FUNCTION_BLOCK FB_FileRingBufferToDB
VAR_INPUT
	udiNovRam_BufferIndex:UDINT;
	udiFile_Index:UDINT;
	dataType:DINT;
END_VAR
VAR_IN_OUT
	NovRamData:ST_NovRam;
END_VAR

IF dataType = E_DB_StructureType.AlarmHistory THEN
	M_AlarmHistory(udiNovRam_BufferIndex:=udiNovRam_BufferIndex,udiFile_Index:=udiFile_Index);
ELSIF dataType = E_DB_StructureType.ProductionHistory THEN
	M_ProductionHistory(udiNovRam_BufferIndex:=udiNovRam_BufferIndex,udiFile_Index:=udiFile_Index);
ELSIF dataType = E_DB_StructureType.ProductionReport THEN
	M_ProductionReport(udiNovRam_BufferIndex:=udiNovRam_BufferIndex,udiFile_Index:=udiFile_Index);
ELSIF dataType = E_DB_StructureType.ProductionSummary THEN
	M_ProductionSummary(udiNovRam_BufferIndex:=udiNovRam_BufferIndex,udiFile_Index:=udiFile_Index);
ELSIF dataType = E_DB_StructureType.SoDuration THEN
	M_SoDuration(udiNovRam_BufferIndex:=udiNovRam_BufferIndex,udiFile_Index:=udiFile_Index);
ELSIF dataType = E_DB_StructureType.StopCount THEN
	M_StopCount(udiNovRam_BufferIndex:=udiNovRam_BufferIndex,udiFile_Index:=udiFile_Index);
ELSIF dataType = E_DB_StructureType.RegularCheckResults THEN
	M_RegularCheckResults(udiNovRam_BufferIndex:=udiNovRam_BufferIndex,udiFile_Index:=udiFile_Index);
END_IF

METHOD M_AlarmHistory : BOOL
VAR_INPUT
	
	//udiFileNo:UDINT;
	udiNovRam_BufferIndex:UDINT;
	udiFile_Index:UDINT;
END_VAR
VAR_INST
	arrDataFromFile:ARRAY[0..GVL.arrArrayLength[E_DB_StructureType.AlarmHistory]-1] OF ST_AlarmInfo_DB_save;//small
	DataToDB:ST_AlarmInfo_DB;//large
	AnalizeIndex:UDINT;//should be kept by NovRam
	iStep:INT;
	i:UDINT;
	fbFileRingBuffer: FB_FileRingBuffer := ( sNetId     := '',
                                             sPathName  := '',
                                             ePath      := PATH_GENERIC,
                                             nID        := 1,
                                             cbBuffer   := gvl.arrFileRingBufferSize[E_DB_StructureType.AlarmHistory], //5MB(5*10^6Bytes)
                                             bOverwrite := FALSE,
                                             pWriteBuff := 0,
                                             cbWriteLen := 0,
                                             pReadBuff  := 0,
                                             cbReadLen  := 0,
                                             tTimeout   := T#1S );
	bBusy:BOOL;
	bError:BOOL;
	nErrID:UDINT;
	stHeader:ST_FileRBufferHead;
    //loadData  : ARRAY[0..511] OF BYTE :=[512(0)];
    //cbLoad    : UDINT;
	
	fileName: STRING(255);
	eStrIndex:DINT;
	fbAlarmHistory_DB		: FB_AlarmHistory_DB;
END_VAR
//Config
eStrIndex:=E_DB_StructureType.AlarmHistory;

fbFileRingBuffer(sPathName:=fileName
				,bBusy=>bBusy,bError=>bError,nErrID=>nErrID
				,stHeader=>stHeader);
//DB_Test
fbAlarmHistory_DB(udiDBID:=1);

CASE iStep OF
	0://check if file full 
		IF NovRamData.arrFileRingBuffer_Status[eStrIndex].bFileFull[udiNovRam_BufferIndex][udiFile_Index] = TRUE//file full = should work 
		THEN
			
			fileName:=M_GetFileName(structureType:=eStrIndex
									,udiNovRam_BufferIndex:=udiNovRam_BufferIndex
									,udiFile_Index:=udiFile_Index);
			
			iStep:=100;
		END_IF
	100:// Open file
		
		AnalizeIndex:=0;
		fbFileRingBuffer.A_Open();
		
		iStep:=200;
	200://wait done / read head
		IF NOT fbFileRingBuffer.bBusy AND NOT fbFileRingBuffer.bError THEN
			
			fbFileRingBuffer.A_GetHead(pReadBuff := ADR(arrDataFromFile), cbReadLen := SIZEOF(arrDataFromFile));
			
			iStep:=300;
		END_IF
	300://wait done / take data from array
		IF NOT fbFileRingBuffer.bBusy AND NOT fbFileRingBuffer.bError THEN
			
			M_ST_AlarmHistory_Extract(Input:=arrDataFromFile[AnalizeIndex],Output=>DataToDB);
			//DataToDB:=arrDataFromFile[AnalizeIndex];
			
			iStep:=310;
		ELSIF NOT fbFileRingBuffer.bBusy AND fbFileRingBuffer.bError THEN//Empty
			iStep:=600;
		END_IF
	310:// write to DB
	
		IF fbAlarmHistory_DB.M_Upload(stAlarmInfo:=DataToDB) THEN
			iStep:=320;
		END_IF
		
	320://wait done
		
		IF NOT fbAlarmHistory_DB.bError THEN//write OK
		
			AnalizeIndex:=AnalizeIndex+1;
			
			iStep:=330;
			
		ELSE//write failed need to write to log
			;
		END_IF
		
	330://Check if all data in array Analized
		IF AnalizeIndex < GVL.arrArrayLength[eStrIndex]-1 THEN//not done
			iStep:=300;//go back
		ELSE//array data done
			iStep:=400;//complete this array
		END_IF
		
	400://wait done / remove Head
	
		fbFileRingBuffer.A_RemoveHead(pReadBuff := ADR(arrDataFromFile), cbReadLen := SIZEOF(arrDataFromFile));
		
		iStep:=500;
		
	500://wait done / check if all data got?
		IF NOT fbFileRingBuffer.bBusy AND NOT fbFileRingBuffer.bError THEN
			IF stHeader.nCount > 0 THEN
				iStep:=100;//Go Back
			ELSE
				iStep:=600;//finish
			END_IF
		END_IF
	600://reset file
	
		fbFileRingBuffer.A_Reset();
		
		iStep:=700;
		
	700://wait done / close file
		IF NOT fbFileRingBuffer.bBusy AND NOT fbFileRingBuffer.bError THEN
			
			fbFileRingBuffer.A_Close();
			
			iStep:=800;
		END_IF
	800://wait done
		IF NOT fbFileRingBuffer.bBusy AND NOT fbFileRingBuffer.bError THEN
			
			NovRamData.arrFileRingBuffer_Status[eStrIndex].bFileFull[udiNovRam_BufferIndex][udiFile_Index]:=FALSE;
			
			iStep:=0;
			
		END_IF
		
	
END_CASE
END_METHOD

METHOD M_GetFileName : STRING(255)
VAR_INPUT
	structureType:DINT;
	udiNovRam_BufferIndex:UDINT;
	udiFile_Index:UDINT;
END_VAR
VAR
	tempString:STRING(255);
	tempString2:STRING(255);
	tempFileNo:UDINT;
END_VAR
IF structureType=E_DB_StructureType.AlarmHistory THEN
	tempString:=CONCAT(gvl.arrfileFolder[structureType],'AlarmHistory');
ELSIF structureType=E_DB_StructureType.ProductionHistory THEN
	tempString:=CONCAT(gvl.arrfileFolder[structureType],'ProductionHistory');
ELSIF structureType=E_DB_StructureType.ProductionReport THEN
	tempString:=CONCAT(gvl.arrfileFolder[structureType],'ProductionReport');
ELSIF structureType=E_DB_StructureType.ProductionSummary THEN
	tempString:=CONCAT(gvl.arrfileFolder[structureType],'ProductionSummary');
ELSIF structureType=E_DB_StructureType.SoDuration THEN
	tempString:=CONCAT(gvl.arrfileFolder[structureType],'SoDuration');
ELSIF structureType=E_DB_StructureType.StopCount THEN
	tempString:=CONCAT(gvl.arrfileFolder[structureType],'StopCount');
ELSIF structureType=E_DB_StructureType.RegularCheckResults THEN
	tempString:=CONCAT(gvl.arrfileFolder[structureType],'RegularCheckResults');
END_IF

tempFileNo:=(udiNovRam_BufferIndex) * GVL.FileRingBufferRatio + (udiFile_Index + 1);
tempString2:=CONCAT(tempString,UDINT_TO_STRING(tempFileNo));
M_GetFileName:=CONCAT(tempString2,'.dat');
END_METHOD

{warning 'add method implementation '}
METHOD M_ProductionHistory : BOOL
VAR_INPUT
	
	//udiFileNo:UDINT;
	udiNovRam_BufferIndex:UDINT;
	udiFile_Index:UDINT;
END_VAR
VAR_INST
	arrDataFromFile:ARRAY[0..GVL.arrArrayLength[E_DB_StructureType.ProductionHistory]-1] OF ST_PHI_GroupData_DB;//small
	DataToDB:ST_PHI_GroupData_DB;//large
	AnalizeIndex:UDINT;//should be kept by NovRam
	iStep:INT;
	i:UDINT;
	fbFileRingBuffer: FB_FileRingBuffer := ( sNetId     := '',
                                             sPathName  := '',
                                             ePath      := PATH_GENERIC,
                                             nID        := 1,
                                             cbBuffer   := gvl.arrFileRingBufferSize[E_DB_StructureType.ProductionHistory], //5MB(5*10^6Bytes)
                                             bOverwrite := FALSE,
                                             pWriteBuff := 0,
                                             cbWriteLen := 0,
                                             pReadBuff  := 0,
                                             cbReadLen  := 0,
                                             tTimeout   := T#1S );
	bBusy:BOOL;
	bError:BOOL;
	nErrID:UDINT;
	stHeader:ST_FileRBufferHead;
    //loadData  : ARRAY[0..511] OF BYTE :=[512(0)];
    //cbLoad    : UDINT;
	
	fileName: STRING(255);
	eStrIndex:DINT;
	
	//DB
	fbProductionHistoryInspection_DB		: FB_ProductionHistoryInspection_DB;
	PHI_GroupData_DB : ST_PHI_GroupData_DB;
END_VAR
//Config
eStrIndex:=E_DB_StructureType.ProductionHistory;

fbFileRingBuffer(sPathName:=fileName
				,bBusy=>bBusy,bError=>bError,nErrID=>nErrID
				,stHeader=>stHeader);
				
//DB_Test
fbProductionHistoryInspection_DB(udiDBID:=1);

CASE iStep OF
	0://check if file full 
		IF NovRamData.arrFileRingBuffer_Status[eStrIndex].bFileFull[udiNovRam_BufferIndex][udiFile_Index] = TRUE//file full = should work 
		THEN
			
			fileName:=M_GetFileName(structureType:=eStrIndex
									,udiNovRam_BufferIndex:=udiNovRam_BufferIndex
									,udiFile_Index:=udiFile_Index);
			
			iStep:=100;
		END_IF
	100:// Open file
		
		AnalizeIndex:=0;
		fbFileRingBuffer.A_Open();
		
		iStep:=200;
	200://wait done / read head
		IF NOT fbFileRingBuffer.bBusy AND NOT fbFileRingBuffer.bError THEN
			
			fbFileRingBuffer.A_GetHead(pReadBuff := ADR(arrDataFromFile), cbReadLen := SIZEOF(arrDataFromFile));
			
			iStep:=300;
		END_IF
	300://wait done / take data from array
		IF NOT fbFileRingBuffer.bBusy AND NOT fbFileRingBuffer.bError THEN
			
			M_ST_ProductionHistory_Extract(Input:=arrDataFromFile[AnalizeIndex],Output=>DataToDB);
			//DataToDB:=arrDataFromFile[AnalizeIndex];
			
			iStep:=310;
		ELSIF NOT fbFileRingBuffer.bBusy AND fbFileRingBuffer.bError THEN//Empty
			iStep:=600;
		END_IF
	310:// write to DB
	
		IF fbProductionHistoryInspection_DB.M_Upload(stPHI:=DataToDB) THEN
			iStep:=320;
		END_IF
		
	320://wait done
		
		IF NOT fbProductionHistoryInspection_DB.bError THEN//write OK
		
			AnalizeIndex:=AnalizeIndex+1;
			
			iStep:=330;
			
		ELSE//write failed need to write to log
			;
		END_IF
		
	330://Check if all data in array Analized
		IF AnalizeIndex < GVL.arrArrayLength[eStrIndex]-1 THEN//not done
			iStep:=300;//go back
		ELSE//array data done
			iStep:=400;//complete this array
		END_IF
		
	400://wait done / remove Head
	
		fbFileRingBuffer.A_RemoveHead(pReadBuff := ADR(arrDataFromFile), cbReadLen := SIZEOF(arrDataFromFile));
		
		iStep:=500;
		
	500://wait done / check if all data got?
		IF NOT fbFileRingBuffer.bBusy AND NOT fbFileRingBuffer.bError THEN
			IF stHeader.nCount > 0 THEN
				iStep:=100;//Go Back
			ELSE
				iStep:=600;//finish
			END_IF
		END_IF
	600://reset file
	
		fbFileRingBuffer.A_Reset();
		
		iStep:=700;
		
	700://wait done / close file
		IF NOT fbFileRingBuffer.bBusy AND NOT fbFileRingBuffer.bError THEN
			
			fbFileRingBuffer.A_Close();
			
			iStep:=800;
		END_IF
	800://wait done
		IF NOT fbFileRingBuffer.bBusy AND NOT fbFileRingBuffer.bError THEN
			
			NovRamData.arrFileRingBuffer_Status[eStrIndex].bFileFull[udiNovRam_BufferIndex][udiFile_Index]:=FALSE;
			
			iStep:=0;
			
		END_IF
		
	
END_CASE
END_METHOD

METHOD M_ProductionReport : BOOL
VAR_INPUT
	
	//udiFileNo:UDINT;
	udiNovRam_BufferIndex:UDINT;
	udiFile_Index:UDINT;
END_VAR
VAR_INST
	arrDataFromFile:ARRAY[0..GVL.arrArrayLength[E_DB_StructureType.ProductionReport]-1] OF ST_OEE_ProductionReport;//small
	DataToDB:ST_OEE_ProductionReport;//large
	AnalizeIndex:UDINT;//should be kept by NovRam
	iStep:INT;
	i:UDINT;
	fbFileRingBuffer: FB_FileRingBuffer := ( sNetId     := '',
                                             sPathName  := '',
                                             ePath      := PATH_GENERIC,
                                             nID        := 1,
                                             cbBuffer   := gvl.arrFileRingBufferSize[E_DB_StructureType.ProductionReport], //5MB(5*10^6Bytes)
                                             bOverwrite := FALSE,
                                             pWriteBuff := 0,
                                             cbWriteLen := 0,
                                             pReadBuff  := 0,
                                             cbReadLen  := 0,
                                             tTimeout   := T#1S );
	bBusy:BOOL;
	bError:BOOL;
	nErrID:UDINT;
	stHeader:ST_FileRBufferHead;
    //loadData  : ARRAY[0..511] OF BYTE :=[512(0)];
    //cbLoad    : UDINT;
	
	fileName: STRING(255);
	eStrIndex:DINT;
	fbOEE_ProductionReport_DB:FB_OEE_ProductionReport_DB;
END_VAR
//Config
eStrIndex:=E_DB_StructureType.ProductionReport;

fbFileRingBuffer(sPathName:=fileName
				,bBusy=>bBusy,bError=>bError,nErrID=>nErrID
				,stHeader=>stHeader);
				
CASE iStep OF
	0://check if file full 
		IF NovRamData.arrFileRingBuffer_Status[eStrIndex].bFileFull[udiNovRam_BufferIndex][udiFile_Index] = TRUE//file full = should work 
		THEN
			
			fileName:=M_GetFileName(structureType:=eStrIndex
									,udiNovRam_BufferIndex:=udiNovRam_BufferIndex
									,udiFile_Index:=udiFile_Index);
			
			iStep:=100;
		END_IF
	100:// Open file
		
		AnalizeIndex:=0;
		fbFileRingBuffer.A_Open();
		
		iStep:=200;
	200://wait done / read head
		IF NOT fbFileRingBuffer.bBusy AND NOT fbFileRingBuffer.bError THEN
			
			fbFileRingBuffer.A_GetHead(pReadBuff := ADR(arrDataFromFile), cbReadLen := SIZEOF(arrDataFromFile));
			
			iStep:=300;
		END_IF
	300://wait done / take data from array
		IF NOT fbFileRingBuffer.bBusy AND NOT fbFileRingBuffer.bError THEN
			
			M_ST_ProductionReport_Extract(Input:=arrDataFromFile[AnalizeIndex],Output=>DataToDB);
			//DataToDB:=arrDataFromFile[AnalizeIndex];
			
			iStep:=310;
		ELSIF NOT fbFileRingBuffer.bBusy AND fbFileRingBuffer.bError THEN//Empty
			iStep:=600;
		END_IF
	310:// write to DB
	
		IF fbOEE_ProductionReport_DB.M_Upload(stOeeProductionReport:=DataToDB) THEN
			iStep:=320;
		END_IF
		
	320://wait done
		
			IF NOT fbOEE_ProductionReport_DB.bError THEN//write OK
			
				AnalizeIndex:=AnalizeIndex+1;
				
				iStep:=330;
				
			ELSE//write failed need to write to log
				;
			END_IF
		
		
	330://Check if all data in array Analized
		IF AnalizeIndex < GVL.arrArrayLength[eStrIndex]-1 THEN//not done
			iStep:=300;//go back
		ELSE//array data done
			iStep:=400;//complete this array
		END_IF
		
	400://wait done / remove Head
	
		fbFileRingBuffer.A_RemoveHead(pReadBuff := ADR(arrDataFromFile), cbReadLen := SIZEOF(arrDataFromFile));
		
		iStep:=500;
		
	500://wait done / check if all data got?
		IF NOT fbFileRingBuffer.bBusy AND NOT fbFileRingBuffer.bError THEN
			IF stHeader.nCount > 0 THEN
				iStep:=100;//Go Back
			ELSE
				iStep:=600;//finish
			END_IF
		END_IF
	600://reset file
	
		fbFileRingBuffer.A_Reset();
		
		iStep:=700;
		
	700://wait done / close file
		IF NOT fbFileRingBuffer.bBusy AND NOT fbFileRingBuffer.bError THEN
			
			fbFileRingBuffer.A_Close();
			
			iStep:=800;
		END_IF
	800://wait done
		IF NOT fbFileRingBuffer.bBusy AND NOT fbFileRingBuffer.bError THEN
			
			NovRamData.arrFileRingBuffer_Status[eStrIndex].bFileFull[udiNovRam_BufferIndex][udiFile_Index]:=FALSE;
			
			iStep:=0;
			
		END_IF
		
	
END_CASE
END_METHOD

METHOD M_ProductionSummary : BOOL
VAR_INPUT
	
	//udiFileNo:UDINT;
	udiNovRam_BufferIndex:UDINT;
	udiFile_Index:UDINT;
END_VAR
VAR_INST
	arrDataFromFile:ARRAY[0..GVL.arrArrayLength[E_DB_StructureType.ProductionSummary]-1] OF ST_OEE_ProductionSummary;//small
	DataToDB:ST_OEE_ProductionSummary;//large
	AnalizeIndex:UDINT;//should be kept by NovRam
	iStep:INT;
	i:UDINT;
	fbFileRingBuffer: FB_FileRingBuffer := ( sNetId     := '',
                                             sPathName  := '',
                                             ePath      := PATH_GENERIC,
                                             nID        := 1,
                                             cbBuffer   := gvl.arrFileRingBufferSize[E_DB_StructureType.ProductionSummary], //5MB(5*10^6Bytes)
                                             bOverwrite := FALSE,
                                             pWriteBuff := 0,
                                             cbWriteLen := 0,
                                             pReadBuff  := 0,
                                             cbReadLen  := 0,
                                             tTimeout   := T#1S );
	bBusy:BOOL;
	bError:BOOL;
	nErrID:UDINT;
	stHeader:ST_FileRBufferHead;
    //loadData  : ARRAY[0..511] OF BYTE :=[512(0)];
    //cbLoad    : UDINT;
	
	fileName: STRING(255);
	eStrIndex:DINT;
	fbOEE_ProductionSummary_DB:FB_OEE_ProductionSummary_DB;
END_VAR
//Config
eStrIndex:=E_DB_StructureType.ProductionSummary;

fbFileRingBuffer(sPathName:=fileName
				,bBusy=>bBusy,bError=>bError,nErrID=>nErrID
				,stHeader=>stHeader);
				
CASE iStep OF
	0://check if file full 
		IF NovRamData.arrFileRingBuffer_Status[eStrIndex].bFileFull[udiNovRam_BufferIndex][udiFile_Index] = TRUE//file full = should work 
		THEN
			
			fileName:=M_GetFileName(structureType:=eStrIndex
									,udiNovRam_BufferIndex:=udiNovRam_BufferIndex
									,udiFile_Index:=udiFile_Index);
			
			iStep:=100;
		END_IF
	100:// Open file
		
		AnalizeIndex:=0;
		fbFileRingBuffer.A_Open();
		
		iStep:=200;
	200://wait done / read head
		IF NOT fbFileRingBuffer.bBusy AND NOT fbFileRingBuffer.bError THEN
			
			fbFileRingBuffer.A_GetHead(pReadBuff := ADR(arrDataFromFile), cbReadLen := SIZEOF(arrDataFromFile));
			
			iStep:=300;
		END_IF
	300://wait done / take data from array
		IF NOT fbFileRingBuffer.bBusy AND NOT fbFileRingBuffer.bError THEN
			
			M_ST_ProductionSummary_Extract(Input:=arrDataFromFile[AnalizeIndex],Output=>DataToDB);
			//DataToDB:=arrDataFromFile[AnalizeIndex];
			
			iStep:=310;
		ELSIF NOT fbFileRingBuffer.bBusy AND fbFileRingBuffer.bError THEN//Empty
			iStep:=600;
		END_IF
	310:// write to DB
	
		IF fbOEE_ProductionSummary_DB.M_Upload(stOEEProductionSummary:=DataToDB) THEN
			iStep:=320;
		END_IF
		
	320://wait done
		
			IF NOT fbOEE_ProductionSummary_DB.bError THEN//write OK
			
				AnalizeIndex:=AnalizeIndex+1;
				
				iStep:=330;
				
			ELSE//write failed need to write to log
				;
			END_IF
		
		
	330://Check if all data in array Analized
		IF AnalizeIndex < GVL.arrArrayLength[eStrIndex]-1 THEN//not done
			iStep:=300;//go back
		ELSE//array data done
			iStep:=400;//complete this array
		END_IF
		
	400://wait done / remove Head
	
		fbFileRingBuffer.A_RemoveHead(pReadBuff := ADR(arrDataFromFile), cbReadLen := SIZEOF(arrDataFromFile));
		
		iStep:=500;
		
	500://wait done / check if all data got?
		IF NOT fbFileRingBuffer.bBusy AND NOT fbFileRingBuffer.bError THEN
			IF stHeader.nCount > 0 THEN
				iStep:=100;//Go Back
			ELSE
				iStep:=600;//finish
			END_IF
		END_IF
	600://reset file
	
		fbFileRingBuffer.A_Reset();
		
		iStep:=700;
		
	700://wait done / close file
		IF NOT fbFileRingBuffer.bBusy AND NOT fbFileRingBuffer.bError THEN
			
			fbFileRingBuffer.A_Close();
			
			iStep:=800;
		END_IF
	800://wait done
		IF NOT fbFileRingBuffer.bBusy AND NOT fbFileRingBuffer.bError THEN
			
			NovRamData.arrFileRingBuffer_Status[eStrIndex].bFileFull[udiNovRam_BufferIndex][udiFile_Index]:=FALSE;
			
			iStep:=0;
			
		END_IF
		
	
END_CASE
END_METHOD

METHOD M_RegularCheckResults : BOOL
VAR_INPUT
	
	//udiFileNo:UDINT;
	udiNovRam_BufferIndex:UDINT;
	udiFile_Index:UDINT;
END_VAR
VAR_INST
	arrDataFromFile:ARRAY[0..GVL.arrArrayLength[E_DB_StructureType.RegularCheckResults]-1] OF ST_RegularCheck_Results;//small
	DataToDB:ST_RegularCheck_Results;//large
	AnalizeIndex:UDINT;//should be kept by NovRam
	iStep:INT;
	i:UDINT;
	fbFileRingBuffer: FB_FileRingBuffer := ( sNetId     := '',
                                             sPathName  := '',
                                             ePath      := PATH_GENERIC,
                                             nID        := 1,
                                             cbBuffer   := gvl.arrFileRingBufferSize[E_DB_StructureType.RegularCheckResults], //5MB(5*10^6Bytes)
                                             bOverwrite := FALSE,
                                             pWriteBuff := 0,
                                             cbWriteLen := 0,
                                             pReadBuff  := 0,
                                             cbReadLen  := 0,
                                             tTimeout   := T#1S );
	bBusy:BOOL;
	bError:BOOL;
	nErrID:UDINT;
	stHeader:ST_FileRBufferHead;
    //loadData  : ARRAY[0..511] OF BYTE :=[512(0)];
    //cbLoad    : UDINT;
	
	fileName: STRING(255);
	eStrIndex:DINT;
	fbRegular_Check_Results_DB:FB_Regular_Check_Results_DB;
END_VAR
//Config
eStrIndex:=E_DB_StructureType.RegularCheckResults;

fbFileRingBuffer(sPathName:=fileName
				,bBusy=>bBusy,bError=>bError,nErrID=>nErrID
				,stHeader=>stHeader);
				
CASE iStep OF
	0://check if file full 
		IF NovRamData.arrFileRingBuffer_Status[eStrIndex].bFileFull[udiNovRam_BufferIndex][udiFile_Index] = TRUE//file full = should work 
		THEN
			
			fileName:=M_GetFileName(structureType:=eStrIndex
									,udiNovRam_BufferIndex:=udiNovRam_BufferIndex
									,udiFile_Index:=udiFile_Index);
			
			iStep:=100;
		END_IF
	100:// Open file
		
		AnalizeIndex:=0;
		fbFileRingBuffer.A_Open();
		
		iStep:=200;
	200://wait done / read head
		IF NOT fbFileRingBuffer.bBusy AND NOT fbFileRingBuffer.bError THEN
			
			fbFileRingBuffer.A_GetHead(pReadBuff := ADR(arrDataFromFile), cbReadLen := SIZEOF(arrDataFromFile));
			
			iStep:=300;
		END_IF
	300://wait done / take data from array
		IF NOT fbFileRingBuffer.bBusy AND NOT fbFileRingBuffer.bError THEN
			
			M_ST_RegularCheckResults_Extract(Input:=arrDataFromFile[AnalizeIndex],Output=>DataToDB);
			//DataToDB:=arrDataFromFile[AnalizeIndex];
								
			iStep:=310;
		ELSIF NOT fbFileRingBuffer.bBusy AND fbFileRingBuffer.bError THEN//Empty
			iStep:=600;
		END_IF
	310:// write to DB
		
		IF fbRegular_Check_Results_DB.M_Upload(stRcResults:=DataToDB) THEN
			iStep:=320;
		END_IF
		
	320://wait done
		
		IF NOT fbRegular_Check_Results_DB.bError THEN//write OK
		
			AnalizeIndex:=AnalizeIndex+1;
			
			iStep:=330;
			
		ELSE//write failed need to write to log
			;
		END_IF
		
	330://Check if all data in array Analized
		IF AnalizeIndex < GVL.arrArrayLength[eStrIndex]-1 THEN//not done
			iStep:=300;//go back
		ELSE//array data done
			iStep:=400;//complete this array
		END_IF
		
	400://wait done / remove Head
	
		fbFileRingBuffer.A_RemoveHead(pReadBuff := ADR(arrDataFromFile), cbReadLen := SIZEOF(arrDataFromFile));
		
		iStep:=500;
		
	500://wait done / check if all data got?
		IF NOT fbFileRingBuffer.bBusy AND NOT fbFileRingBuffer.bError THEN
			IF stHeader.nCount > 0 THEN
				iStep:=100;//Go Back
			ELSE
				iStep:=600;//finish
			END_IF
		END_IF
	600://reset file
	
		fbFileRingBuffer.A_Reset();
		
		iStep:=700;
		
	700://wait done / close file
		IF NOT fbFileRingBuffer.bBusy AND NOT fbFileRingBuffer.bError THEN
			
			fbFileRingBuffer.A_Close();
			
			iStep:=800;
		END_IF
	800://wait done
		IF NOT fbFileRingBuffer.bBusy AND NOT fbFileRingBuffer.bError THEN
			
			NovRamData.arrFileRingBuffer_Status[eStrIndex].bFileFull[udiNovRam_BufferIndex][udiFile_Index]:=FALSE;
			
			iStep:=0;
			
		END_IF
		
	
END_CASE
END_METHOD

METHOD M_SoDuration : BOOL
VAR_INPUT
	
	//udiFileNo:UDINT;
	udiNovRam_BufferIndex:UDINT;
	udiFile_Index:UDINT;
END_VAR
VAR_INST
	arrDataFromFile:ARRAY[0..GVL.arrArrayLength[E_DB_StructureType.SoDuration]-1] OF ST_SoDuration;//small
	DataToDB:ST_SoDuration;//large
	AnalizeIndex:UDINT;//should be kept by NovRam
	iStep:INT;
	i:UDINT;
	fbFileRingBuffer: FB_FileRingBuffer := ( sNetId     := '',
                                             sPathName  := '',
                                             ePath      := PATH_GENERIC,
                                             nID        := 1,
                                             cbBuffer   := gvl.arrFileRingBufferSize[E_DB_StructureType.ProductionSummary], //5MB(5*10^6Bytes)
                                             bOverwrite := FALSE,
                                             pWriteBuff := 0,
                                             cbWriteLen := 0,
                                             pReadBuff  := 0,
                                             cbReadLen  := 0,
                                             tTimeout   := T#1S );
	bBusy:BOOL;
	bError:BOOL;
	nErrID:UDINT;
	stHeader:ST_FileRBufferHead;
    //loadData  : ARRAY[0..511] OF BYTE :=[512(0)];
    //cbLoad    : UDINT;
	
	fileName: STRING(255);
	eStrIndex:DINT;
	fbSoDuration_DB:FB_SoDuration_DB;
	
END_VAR
//Config
eStrIndex:=E_DB_StructureType.SoDuration;

fbFileRingBuffer(sPathName:=fileName
				,bBusy=>bBusy,bError=>bError,nErrID=>nErrID
				,stHeader=>stHeader);
				
CASE iStep OF
	0://check if file full 
		IF NovRamData.arrFileRingBuffer_Status[eStrIndex].bFileFull[udiNovRam_BufferIndex][udiFile_Index] = TRUE//file full = should work 
		THEN
			
			fileName:=M_GetFileName(structureType:=eStrIndex
									,udiNovRam_BufferIndex:=udiNovRam_BufferIndex
									,udiFile_Index:=udiFile_Index);
			
			iStep:=100;
		END_IF
	100:// Open file
		
		AnalizeIndex:=0;
		fbFileRingBuffer.A_Open();
		
		iStep:=200;
	200://wait done / read head
		IF NOT fbFileRingBuffer.bBusy AND NOT fbFileRingBuffer.bError THEN
			
			fbFileRingBuffer.A_GetHead(pReadBuff := ADR(arrDataFromFile), cbReadLen := SIZEOF(arrDataFromFile));
			
			iStep:=300;
		END_IF
	300://wait done / take data from array
		IF NOT fbFileRingBuffer.bBusy AND NOT fbFileRingBuffer.bError THEN
			
			M_ST_SoDuration_Extract(Input:=arrDataFromFile[AnalizeIndex],Output=>DataToDB);
			//DataToDB:=arrDataFromFile[AnalizeIndex];
			
			iStep:=310;
		ELSIF NOT fbFileRingBuffer.bBusy AND fbFileRingBuffer.bError THEN//Empty
			iStep:=600;
		END_IF
	310:// write to DB
	
		IF fbSoDuration_DB.M_Upload(stSoDuration:=DataToDB) THEN
			iStep:=320;
		END_IF
		
	320://wait done
		
		IF NOT fbSoDuration_DB.bError THEN//write OK
		
			AnalizeIndex:=AnalizeIndex+1;
			
			iStep:=330;
			
		ELSE//write failed need to write to log
			;
		END_IF
		
	330://Check if all data in array Analized
		IF AnalizeIndex < GVL.arrArrayLength[eStrIndex]-1 THEN//not done
			iStep:=300;//go back
		ELSE//array data done
			iStep:=400;//complete this array
		END_IF
		
	400://wait done / remove Head
	
		fbFileRingBuffer.A_RemoveHead(pReadBuff := ADR(arrDataFromFile), cbReadLen := SIZEOF(arrDataFromFile));
		
		iStep:=500;
		
	500://wait done / check if all data got?
		IF NOT fbFileRingBuffer.bBusy AND NOT fbFileRingBuffer.bError THEN
			IF stHeader.nCount > 0 THEN
				iStep:=100;//Go Back
			ELSE
				iStep:=600;//finish
			END_IF
		END_IF
	600://reset file
	
		fbFileRingBuffer.A_Reset();
		
		iStep:=700;
		
	700://wait done / close file
		IF NOT fbFileRingBuffer.bBusy AND NOT fbFileRingBuffer.bError THEN
			
			fbFileRingBuffer.A_Close();
			
			iStep:=800;
		END_IF
	800://wait done
		IF NOT fbFileRingBuffer.bBusy AND NOT fbFileRingBuffer.bError THEN
			
			NovRamData.arrFileRingBuffer_Status[eStrIndex].bFileFull[udiNovRam_BufferIndex][udiFile_Index]:=FALSE;
			
			iStep:=0;
			
		END_IF
		
	
END_CASE
END_METHOD

METHOD M_ST_AlarmHistory_Extract : BOOL
VAR_INPUT
	Input:ST_AlarmInfo_DB_save;
END_VAR
VAR_OUTPUT
	Output:ST_AlarmInfo_DB;
END_VAR
Output.lrTime_ms:=Input.lrTime_ms;
Output.iMsgProc:=Input.iMsgProc;
Output.iStateAfter:=Input.iStateAfter;
Output.iMsgClass:=Input.iMsgClass;
Output.diMsgNumber:=Input.diMsgNumber;
Output.sTimeString:=Input.sTimeString;
Output.wsMsgText:=Input.wsMsgText;
Output.sPLC:=Input.sPLC;
Output.wsEquipment:=Input.wsEquipment;
Output.sFaam_id:=Input.sFaam_id;
END_METHOD

METHOD M_ST_ProductionHistory_Extract : BOOL
VAR_INPUT
	Input:ST_PHI_GroupData_DB;
END_VAR
VAR_OUTPUT
	Output:ST_PHI_GroupData_DB;
END_VAR
Output:=Input;
END_METHOD

METHOD M_ST_ProductionReport_Extract : BOOL
VAR_INPUT
	Input:ST_OEE_ProductionReport;
END_VAR
VAR_OUTPUT
	Output:ST_OEE_ProductionReport;
END_VAR
Output:=Input;
END_METHOD

METHOD M_ST_ProductionSummary_Extract : BOOL
VAR_INPUT
	Input:ST_OEE_ProductionSummary;
END_VAR
VAR_OUTPUT
	Output:ST_OEE_ProductionSummary;
END_VAR
Output:=Input;
END_METHOD

METHOD M_ST_RegularCheckResults_Extract : BOOL
VAR_INPUT
	Input:ST_RegularCheck_Results;
END_VAR
VAR_OUTPUT
	Output:ST_RegularCheck_Results;
END_VAR
(*
Output.diStation_number:=Input.diStation_number;
Output.diTrack_number:=Input.diTrack_number;
Output.dtStart_time:=Input.dtStart_time;

IF Input.eSensor = E_RegularCheckSensorResult.Pass THEN
	Output.bSensor:=TRUE;
ELSE
	Output.bSensor:=FALSE;
END_IF

IF Input.eCamera = E_RegularCheckSensorResult.Pass THEN
	Output.bCamera:=TRUE;
ELSE
	Output.bCamera:=FALSE;
END_IF

IF Input.eLoadcell = E_RegularCheckSensorResult.Pass THEN
	Output.bLoadcell:=TRUE;
ELSE
	Output.bLoadcell:=FALSE;
END_IF

IF Input.eSensor2 = E_RegularCheckSensorResult.Pass THEN
	Output.bSensor2:=TRUE;
ELSE
	Output.bSensor2:=FALSE;
END_IF

Output.diRegular_check_id:=Input.diRegular_check_id;
Output.sFaam_id:=Input.sFaam_id;
Output.sSo_number:=Input.sSo_number;
Output.diSo_id:=Input.diSo_id;
Output.wsEmployee_name_logged_in:=Input.wsEmployee_name_logged_in;
*)
Output:=Input;
END_METHOD

METHOD M_ST_SoDuration_Extract : BOOL
VAR_INPUT
	Input:ST_SoDuration;
END_VAR
VAR_OUTPUT
	Output:ST_SoDuration;
END_VAR
Output:=Input;
END_METHOD

METHOD M_ST_StopCount_Extract : BOOL
VAR_INPUT
	Input:ST_StopCount;
END_VAR
VAR_OUTPUT
	Output:ST_StopCount;
END_VAR
Output:=Input;
END_METHOD

METHOD M_StopCount : BOOL
VAR_INPUT
	
	//udiFileNo:UDINT;
	udiNovRam_BufferIndex:UDINT;
	udiFile_Index:UDINT;
END_VAR
VAR_INST
	arrDataFromFile:ARRAY[0..GVL.arrArrayLength[E_DB_StructureType.StopCount]-1] OF ST_StopCount;//small
	DataToDB:ST_StopCount;//large
	AnalizeIndex:UDINT;//should be kept by NovRam
	iStep:INT;
	i:UDINT;
	fbFileRingBuffer: FB_FileRingBuffer := ( sNetId     := '',
                                             sPathName  := '',
                                             ePath      := PATH_GENERIC,
                                             nID        := 1,
                                             cbBuffer   := gvl.arrFileRingBufferSize[E_DB_StructureType.StopCount], //5MB(5*10^6Bytes)
                                             bOverwrite := FALSE,
                                             pWriteBuff := 0,
                                             cbWriteLen := 0,
                                             pReadBuff  := 0,
                                             cbReadLen  := 0,
                                             tTimeout   := T#1S );
	bBusy:BOOL;
	bError:BOOL;
	nErrID:UDINT;
	stHeader:ST_FileRBufferHead;
    //loadData  : ARRAY[0..511] OF BYTE :=[512(0)];
    //cbLoad    : UDINT;
	
	fileName: STRING(255);
	eStrIndex:DINT;
	fbStopCount_DB:FB_StopCount_DB;
END_VAR
//Config
eStrIndex:=E_DB_StructureType.StopCount;

fbFileRingBuffer(sPathName:=fileName
				,bBusy=>bBusy,bError=>bError,nErrID=>nErrID
				,stHeader=>stHeader);
				
CASE iStep OF
	0://check if file full 
		IF NovRamData.arrFileRingBuffer_Status[eStrIndex].bFileFull[udiNovRam_BufferIndex][udiFile_Index] = TRUE//file full = should work 
		THEN
			
			fileName:=M_GetFileName(structureType:=eStrIndex
									,udiNovRam_BufferIndex:=udiNovRam_BufferIndex
									,udiFile_Index:=udiFile_Index);
			
			iStep:=100;
		END_IF
	100:// Open file
		
		AnalizeIndex:=0;
		fbFileRingBuffer.A_Open();
		
		iStep:=200;
	200://wait done / read head
		IF NOT fbFileRingBuffer.bBusy AND NOT fbFileRingBuffer.bError THEN
			
			fbFileRingBuffer.A_GetHead(pReadBuff := ADR(arrDataFromFile), cbReadLen := SIZEOF(arrDataFromFile));
			
			iStep:=300;
		END_IF
	300://wait done / take data from array
		IF NOT fbFileRingBuffer.bBusy AND NOT fbFileRingBuffer.bError THEN
			
			M_ST_StopCount_Extract(Input:=arrDataFromFile[AnalizeIndex],Output=>DataToDB);
			//DataToDB:=arrDataFromFile[AnalizeIndex];
			
			iStep:=310;
		ELSIF NOT fbFileRingBuffer.bBusy AND fbFileRingBuffer.bError THEN//Empty
			iStep:=600;
		END_IF
	310:// write to DB
		
		IF fbStopCount_DB.M_Upload(stStopCount:=DataToDB) THEN
			iStep:=320;
		END_IF
		
	320://wait done
		
		IF NOT fbStopCount_DB.bError THEN//write OK
		
			AnalizeIndex:=AnalizeIndex+1;
			
			iStep:=330;
			
		ELSE//write failed need to write to log
			;
		END_IF
		
	330://Check if all data in array Analized
		IF AnalizeIndex < GVL.arrArrayLength[eStrIndex]-1 THEN//not done
			iStep:=300;//go back
		ELSE//array data done
			iStep:=400;//complete this array
		END_IF
		
	400://wait done / remove Head
	
		fbFileRingBuffer.A_RemoveHead(pReadBuff := ADR(arrDataFromFile), cbReadLen := SIZEOF(arrDataFromFile));
		
		iStep:=500;
		
	500://wait done / check if all data got?
		IF NOT fbFileRingBuffer.bBusy AND NOT fbFileRingBuffer.bError THEN
			IF stHeader.nCount > 0 THEN
				iStep:=100;//Go Back
			ELSE
				iStep:=600;//finish
			END_IF
		END_IF
	600://reset file
	
		fbFileRingBuffer.A_Reset();
		
		iStep:=700;
		
	700://wait done / close file
		IF NOT fbFileRingBuffer.bBusy AND NOT fbFileRingBuffer.bError THEN
			
			fbFileRingBuffer.A_Close();
			
			iStep:=800;
		END_IF
	800://wait done
		IF NOT fbFileRingBuffer.bBusy AND NOT fbFileRingBuffer.bError THEN
			
			NovRamData.arrFileRingBuffer_Status[eStrIndex].bFileFull[udiNovRam_BufferIndex][udiFile_Index]:=FALSE;
			
			iStep:=0;
			
		END_IF
		
	
END_CASE
END_METHOD

END_FUNCTION_BLOCK

(* stored: Version 1.1.0.1, ProductVersion 3.1.4024.11
   POU FB_FileRingBufferToDB: Id {5407df28-5241-4688-9419-685e8c9548d2}, SpecialFunc None
   Folder Sub: Id {99009e46-9b2f-446b-9e3c-ddc566aff4a9}
   Method M_AlarmHistory: Id {ff77384c-01f1-48bd-a1b3-7abc9b26720b}
   Method M_GetFileName: Id {4b3fabe7-1e25-46e4-9798-bee9befa9ab6}
   Method M_ProductionHistory: Id {8fa7d530-7099-445c-bf55-d19dcfd86a46}
   Method M_ProductionReport: Id {50ec54d4-867e-4233-ac7e-27f8467d1362}
   Method M_ProductionSummary: Id {cc4bac99-b6fb-4a33-86fa-fb65566bf866}
   Method M_RegularCheckResults: Id {c1a33c14-6851-44f5-b745-cb1a1bc9c7c4}
   Method M_SoDuration: Id {56393071-2555-404b-aac1-71b9d39a0087}
   Method M_ST_AlarmHistory_Extract: Id {5b8cd87c-96ee-4037-a202-d74d22085ccd}
   Method M_ST_ProductionHistory_Extract: Id {68baffc9-f706-47d6-88f8-4abf8842d603}
   Method M_ST_ProductionReport_Extract: Id {af148257-03fa-4365-8a2d-22bdd2769cf2}
   Method M_ST_ProductionSummary_Extract: Id {b22ff7b2-fb36-43d4-a8ad-c66ee5dbbec5}
   Method M_ST_RegularCheckResults_Extract: Id {01020571-a260-43f0-9306-9b35a4d8ba81}
   Method M_ST_SoDuration_Extract: Id {041093b7-486b-4764-8273-d6a2053f8837}
   Method M_ST_StopCount_Extract: Id {a101ea81-d579-4034-acb4-b6adc3e24537}
   Method M_StopCount: Id {ce4c351f-2ecd-476b-900a-3eebce8b4087} *)
